{attribute 'GeneratedUsingTerminal: '}
{attribute addProperty BoxType ""}
{attribute addProperty Id "_defaultAT %I*SyncUnitTasks_6FEB825718"}
{attribute addProperty CRC "2581955759"}
{attribute addProperty Size "18"}
TYPE SyncUnits_99E584AF :
STRUCT
	{attribute addProperty Name "_default"}
	_default : SyncUnitTasks_6FEB8257;
END_STRUCT
END_TYPE

(* stored: Version 1.2.0.0, ProductVersion 3.1.4024.9
   DUT SyncUnits_99E584AF: Id {a5718ca0-29af-4616-aec0-b68c0605e640} *)
